Yaskawa INFORM job: 04152026.JBI

/JOB
//NAME 04152026
//POS
///NPOS 22,0,0,0,0,0
///TOOL 0
///POSTYPE PULSE
///PULSE
C00000=-2822,58859,-1118,-1041,-34109,-89
C00001=-1968,58778,-1261,-1155,-34032,-431
C00002=-2114,58450,-1762,-1141,-33831,-368
C00003=-2261,58122,-2261,-1127,-33630,-305
C00004=-2406,57791,-2763,-1113,-33428,-243
C00005=-2555,57463,-3262,-1098,-33228,-179
C00006=-2701,57130,-3765,-1084,-33027,-117
C00007=-2852,56800,-4263,-1068,-32828,-52
C00008=-2907,56521,-4684,-1065,-32660,-27
C00009=-2603,56508,-4704,-1106,-32649,-148
C00010=-2299,56494,-4725,-1148,-32637,-269
C00011=-1995,56481,-4745,-1189,-32625,-390
C00012=-1691,56468,-4765,-1230,-32614,-511
C00013=-1387,56454,-4786,-1272,-32603,-632
C00014=-1083,56441,-4806,-1313,-32591,-753
C00015=-1150,56734,-4359,-1299,-32774,-731
C00016=-1288,57074,-3841,-1274,-32985,-680
C00017=-1429,57414,-3325,-1249,-33195,-629
C00018=-1560,57758,-2802,-1226,-33408,-581
C00019=-1698,58100,-2286,-1201,-33618,-531
C00020=-1832,58444,-1766,-1178,-33828,-482
C00021=-1968,58778,-1261,-1155,-34032,-431
//INST
///DATE 2026/04/15 15:34
///ATTR SC,RW
///GROUP1 RB1
NOP
MOVJ C00000 VJ=0.78
MOVJ C00001 VJ=0.78
MOVJ C00002 VJ=0.78
MOVJ C00003 VJ=0.78
MOVJ C00004 VJ=0.78
MOVJ C00005 VJ=0.78
MOVJ C00006 VJ=0.78
MOVJ C00007 VJ=0.78
MOVJ C00008 VJ=0.78
MOVJ C00009 VJ=0.78
MOVJ C00010 VJ=0.78
MOVJ C00011 VJ=0.78
MOVJ C00012 VJ=0.78
MOVJ C00013 VJ=0.78
MOVJ C00014 VJ=0.78
MOVJ C00015 VJ=0.78
MOVJ C00016 VJ=0.78
MOVJ C00017 VJ=0.78
MOVJ C00018 VJ=0.78
MOVJ C00019 VJ=0.78
MOVJ C00020 VJ=0.78
MOVJ C00021 VJ=0.78
END
